// TIA Portal project "Scambio_ferroviario3" (V15.1)

(* hardware
DEVICE "S7-1200 station_1"  S7-1200 Station
   slot 0: "Telaio di montaggio_0"  S7-1200 Rack  Rack  V1.0
   slot 1: "PLC_1"  CPU 1214C DC/DC/DC  6ES7 214-1AG40-0XB0  V4.2
*)

// ===== PLC "PLC_1"  CPU 1214C DC/DC/DC =====

VAR_GLOBAL   // PLC tag table "Tabella delle variabili standard"
   "occupato" AT %M0.0 : Bool;
   "P1" AT %I0.0 : Bool;
   "P2" AT %I0.1 : Bool;
   "SP1" AT %I0.2 : Bool;
   "SP2" AT %I0.3 : Bool;
   "SA1" AT %I0.4 : Bool;
   "SA2" AT %I0.5 : Bool;
   "A" AT %I0.6 : Bool;
   "B" AT %I0.7 : Bool;
   "C" AT %I1.0 : Bool;
   "D" AT %I1.1 : Bool;
   "S1" AT %Q0.0 : Bool;
   "D1" AT %Q0.1 : Bool;
   "S2" AT %Q0.2 : Bool;
   "D2" AT %Q0.3 : Bool;
   "SC1" AT %Q0.4 : Bool;
   "SC2" AT %Q0.5 : Bool;
END_VAR

VAR_GLOBAL CONSTANT   // PLC tag table "Tabella delle variabili standard"
   "TempoAttesa" : Time := T#60s;
END_VAR

DATA_BLOCK "movimento_carrello_DB"   // DB1
{ S7_Optimized_Access := 'TRUE' }
VERSION : 0.1
// stored: InstanceOfName movimento_carrello
"movimento_carrello"
BEGIN
END_DATA_BLOCK

DATA_BLOCK "movimento_carrello_DB_1"   // DB2
{ S7_Optimized_Access := 'TRUE' }
VERSION : 0.1
// stored: InstanceOfName movimento_carrello
"movimento_carrello"
BEGIN
END_DATA_BLOCK

DATA_BLOCK "movimento_carrello_DB_2"   // DB3
{ S7_Optimized_Access := 'TRUE' }
VERSION : 0.1
// stored: InstanceOfName movimento_carrello
"movimento_carrello"
BEGIN
END_DATA_BLOCK

DATA_BLOCK "movimento_carrello_DB_3"   // DB4
{ S7_Optimized_Access := 'TRUE' }
VERSION : 0.1
// stored: InstanceOfName movimento_carrello
"movimento_carrello"
BEGIN
END_DATA_BLOCK

FUNCTION_BLOCK "movimento_carrello"   // FB1, LAD
{ S7_Optimized_Access := 'TRUE' }
VERSION : 0.1
   VAR_INPUT
      partenza : Bool;
      finecorsaPartenza : Bool;
      finecorsaArrivo : Bool;
      finecorsaPrimoScambio : Bool;
      finecorsaSecondoScambio : Bool;
      mode : Bool;
   END_VAR
   VAR_OUTPUT
      scambio1 : Bool;
      scambio2 : Bool;
      motore : Bool;
   END_VAR
   VAR RETAIN
      home : Bool := true;
      muovi1 : Bool;
      attesa : Bool;
      muovi2 : Bool;
      muovi3 : Bool;
   END_VAR
   VAR
      wait : Bool;
      IEC_Timer_0_Instance : TON_TIME;
   END_VAR
BEGIN

REGION Network 1
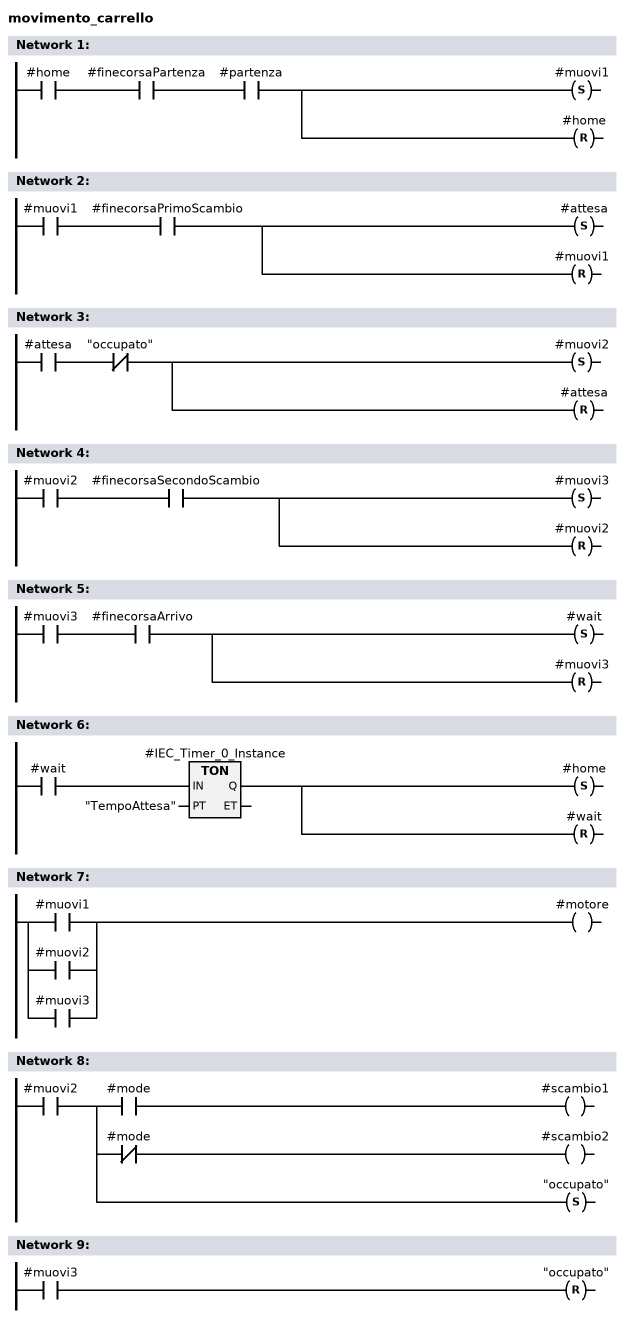
   RUNG wire#powerrail
      Contact( #home )
      Contact( #finecorsaPartenza )
      Contact( #partenza )
      wire#w1
      S_Coil( #muovi1 )
   END_RUNG
   RUNG wire#w1
      R_Coil( #home )
   END_RUNG
   // the same network as SCL:
   IF #home AND #finecorsaPartenza AND #partenza THEN
       #muovi1 := TRUE;
       #home := FALSE;
   END_IF;
END_REGION

REGION Network 2
   RUNG wire#powerrail
      Contact( #muovi1 )
      Contact( #finecorsaPrimoScambio )
      wire#w1
      S_Coil( #attesa )
   END_RUNG
   RUNG wire#w1
      R_Coil( #muovi1 )
   END_RUNG
   // the same network as SCL:
   IF #muovi1 AND #finecorsaPrimoScambio THEN
       #attesa := TRUE;
       #muovi1 := FALSE;
   END_IF;
END_REGION

REGION Network 3
   RUNG wire#powerrail
      Contact( #attesa )
      I_Contact( "occupato" )
      wire#w1
      S_Coil( #muovi2 )
   END_RUNG
   RUNG wire#w1
      R_Coil( #attesa )
   END_RUNG
   // the same network as SCL:
   IF #attesa AND NOT "occupato" THEN
       #muovi2 := TRUE;
       #attesa := FALSE;
   END_IF;
END_REGION

REGION Network 4
   RUNG wire#powerrail
      Contact( #muovi2 )
      Contact( #finecorsaSecondoScambio )
      wire#w1
      S_Coil( #muovi3 )
   END_RUNG
   RUNG wire#w1
      R_Coil( #muovi2 )
   END_RUNG
   // the same network as SCL:
   IF #muovi2 AND #finecorsaSecondoScambio THEN
       #muovi3 := TRUE;
       #muovi2 := FALSE;
   END_IF;
END_REGION

REGION Network 5
   RUNG wire#powerrail
      Contact( #muovi3 )
      Contact( #finecorsaArrivo )
      wire#w1
      S_Coil( #wait )
   END_RUNG
   RUNG wire#w1
      R_Coil( #muovi3 )
   END_RUNG
   // the same network as SCL:
   IF #muovi3 AND #finecorsaArrivo THEN
       #wait := TRUE;
       #muovi3 := FALSE;
   END_IF;
END_REGION

REGION Network 6
   #IEC_Timer_0_Instance(IN := #wait, PT := "TempoAttesa");   // TON
   IF #IEC_Timer_0_Instance.Q THEN
       #home := TRUE;
       #wait := FALSE;
   END_IF;
END_REGION

REGION Network 7
   RUNG wire#powerrail
      Contact( #muovi1 )
      wire#w1
      Coil( #motore )
   END_RUNG
   RUNG wire#powerrail
      Contact( #muovi2 )
   END_RUNG wire#w1
   RUNG wire#powerrail
      Contact( #muovi3 )
   END_RUNG wire#w1
   // the same network as SCL:
   #motore := #muovi1 OR #muovi2 OR #muovi3;
END_REGION

REGION Network 8
   RUNG wire#powerrail
      Contact( #muovi2 )
      wire#w1
      Contact( #mode )
      Coil( #scambio1 )
   END_RUNG
   RUNG wire#w1
      I_Contact( #mode )
      Coil( #scambio2 )
   END_RUNG
   RUNG wire#w1
      S_Coil( "occupato" )
   END_RUNG
   // the same network as SCL:
   #scambio1 := #muovi2 AND #mode;
   #scambio2 := #muovi2 AND NOT #mode;
   IF #muovi2 THEN "occupato" := TRUE; END_IF;
END_REGION

REGION Network 9
   RUNG wire#powerrail
      Contact( #muovi3 )
      R_Coil( "occupato" )
   END_RUNG
   // the same network as SCL:
   IF #muovi3 THEN "occupato" := FALSE; END_IF;
END_REGION
END_FUNCTION_BLOCK

ORGANIZATION_BLOCK "Main"   // OB1, LAD, ProgramCycle
TITLE = "Main Program Sweep (Cycle)"
{ S7_Optimized_Access := 'TRUE' }
VERSION : 0.1
   VAR_INPUT
      Initial_Call : Bool;   // Initial call of this OB
      Remanence : Bool;   // =True, if remanent data are available
   END_VAR
BEGIN

REGION Network 1
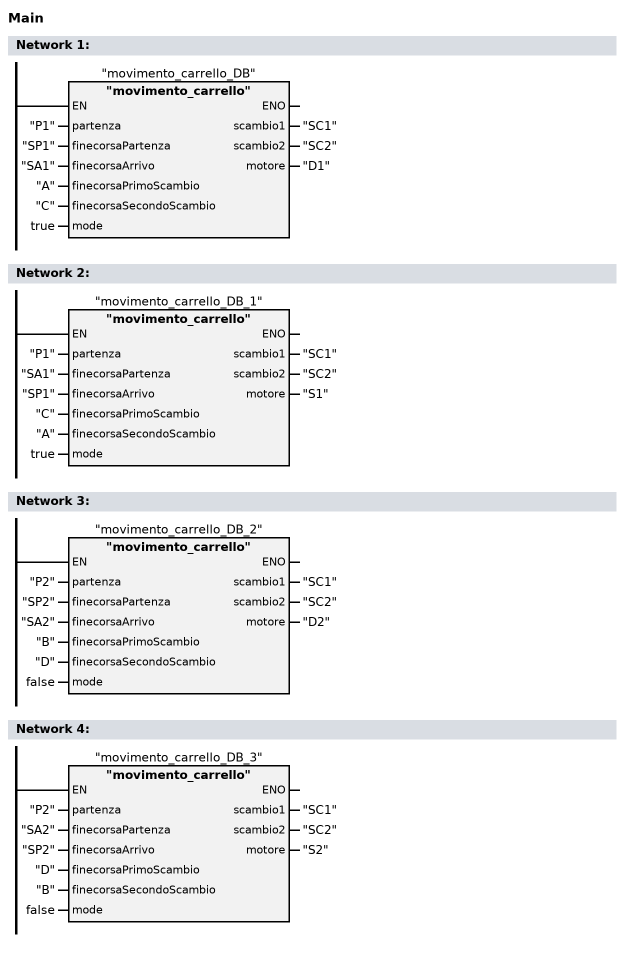
   RUNG wire#powerrail
      "movimento_carrello_DB"(partenza := "P1", finecorsaPartenza := "SP1", finecorsaArrivo := "SA1", finecorsaPrimoScambio := "A", finecorsaSecondoScambio := "C", mode := true, scambio1 => "SC1", scambio2 => "SC2", motore => "D1")
   END_RUNG
   // the same network as SCL:
   "movimento_carrello_DB"(partenza := "P1",   // "movimento_carrello"
                           finecorsaPartenza := "SP1",
                           finecorsaArrivo := "SA1",
                           finecorsaPrimoScambio := "A",
                           finecorsaSecondoScambio := "C",
                           mode := true,
                           scambio1 => "SC1",
                           scambio2 => "SC2",
                           motore => "D1");
END_REGION

REGION Network 2
   RUNG wire#powerrail
      "movimento_carrello_DB_1"(partenza := "P1", finecorsaPartenza := "SA1", finecorsaArrivo := "SP1", finecorsaPrimoScambio := "C", finecorsaSecondoScambio := "A", mode := true, scambio1 => "SC1", scambio2 => "SC2", motore => "S1")
   END_RUNG
   // the same network as SCL:
   "movimento_carrello_DB_1"(partenza := "P1",   // "movimento_carrello"
                           finecorsaPartenza := "SA1",
                           finecorsaArrivo := "SP1",
                           finecorsaPrimoScambio := "C",
                           finecorsaSecondoScambio := "A",
                           mode := true,
                           scambio1 => "SC1",
                           scambio2 => "SC2",
                           motore => "S1");
END_REGION

REGION Network 3
   RUNG wire#powerrail
      "movimento_carrello_DB_2"(partenza := "P2", finecorsaPartenza := "SP2", finecorsaArrivo := "SA2", finecorsaPrimoScambio := "B", finecorsaSecondoScambio := "D", mode := false, scambio1 => "SC1", scambio2 => "SC2", motore => "D2")
   END_RUNG
   // the same network as SCL:
   "movimento_carrello_DB_2"(partenza := "P2",   // "movimento_carrello"
                           finecorsaPartenza := "SP2",
                           finecorsaArrivo := "SA2",
                           finecorsaPrimoScambio := "B",
                           finecorsaSecondoScambio := "D",
                           mode := false,
                           scambio1 => "SC1",
                           scambio2 => "SC2",
                           motore => "D2");
END_REGION

REGION Network 4
   RUNG wire#powerrail
      "movimento_carrello_DB_3"(partenza := "P2", finecorsaPartenza := "SA2", finecorsaArrivo := "SP2", finecorsaPrimoScambio := "D", finecorsaSecondoScambio := "B", mode := false, scambio1 => "SC1", scambio2 => "SC2", motore => "S2")
   END_RUNG
   // the same network as SCL:
   "movimento_carrello_DB_3"(partenza := "P2",   // "movimento_carrello"
                           finecorsaPartenza := "SA2",
                           finecorsaArrivo := "SP2",
                           finecorsaPrimoScambio := "D",
                           finecorsaSecondoScambio := "B",
                           mode := false,
                           scambio1 => "SC1",
                           scambio2 => "SC2",
                           motore => "S2");
END_REGION
END_ORGANIZATION_BLOCK